FUNCTION BitLesen : BOOL
VAR_INPUT
Eingang: BYTE;
	Position: BYTE;
END_VAR
VAR
	Bitmuster: BYTE;
END_VAR

Bitmuster := SHL(1, Position);
IF ((Eingang AND Bitmuster) = Bitmuster) THEN
	BitLesen := TRUE;
ELSE		
	BitLesen:= FALSE;	
END_IF;

END_FUNCTION

(* stored: Version 1.1.0.1, ProductVersion 3.1.4024.5
   POU BitLesen: Id {e6a103b1-82cc-43e6-bec5-7490cb54c7e5}, SpecialFunc None *)
